PROGRAM Main_10ms
VAR
END_VAR


Prg_GetClock();
Prg_logEvents();
OpenExplorer();

END_PROGRAM

(* stored: Version 1.1.0.1, ProductVersion 3.1.4024.13
   POU Main_10ms: Id {29894ea1-65c2-4e7c-956e-9f59c5a57d0c}, SpecialFunc None *)
